FUNCTION_BLOCK FB_ConveyorControl_Test EXTENDS TcUnit.FB_TestSuite
VAR
END_VAR

TestConveyorBuildCheck();

METHOD PRIVATE TestConveyorBuildCheck
VAR
	hmi : ST_ConveyorHMI;
END_VAR
TEST('TestConveyorBuildCheck');

hmi.eSystemStatus := E_ConveyorStatus.Stopped;
hmi.fBeltSpeed := 0.0;
hmi.nTodayCount := 0;

AssertEquals_UINT(Expected := 0, Actual := hmi.eSystemStatus, Message := 'Status should be Stopped');

TEST_FINISHED();
END_METHOD

END_FUNCTION_BLOCK

(* stored: Version 1.1.0.1, ProductVersion 3.1.4026.17
   POU FB_ConveyorControl_Test: Id {1294cbc6-0ada-4602-bf3a-379f7a2047c4}, SpecialFunc None
   Method TestConveyorBuildCheck: Id {0b1332b7-22df-426d-bb42-2723a9680ab8} *)
